// TwinCAT 3 PLC project Untitled1
// ProgramVersion: 3.1.4026.17
// libraries:
//   Tc2_Standard, * (Beckhoff Automation GmbH)
//   Tc2_System, * (Beckhoff Automation GmbH)
//   Tc2_Utilities, * (Beckhoff Automation GmbH)
//   Tc3_EventLogger, * (Beckhoff Automation GmbH)
// project tree:
//   / PlcTask.TcTTO
//   POUs/ Batch.TcPOU, MAIN.TcPOU
// real-time tasks:
//   TASK PlcTask: cycle T#10ms, priority 20, ADS port 350
// I/O:
//   DEVICE Device 2 (EtherCAT) (disabled), AmsNetId 10.12.64.53.3.1
//     Term 1 (EK1100) [EK1100 EtherCAT Coupler (2A E-Bus)]
//       Term 2 (EL1018) [EL1018 8Ch. Dig. Input 24V, 10µs]
//       Term 3 (EL1382) [EL1382 2Ch. Dig. Input thermistor]
//       Term 4 (EL6070-0033) [EL6070-0033 1Ch. Licence key terminal, individual licences]
//       Term 5 (EL6900) [EL6900, TwinSAFE PLC]
//       Term 6 (EL1918) [EL1918, 8Ch. Safety Input 24V, TwinSAFE]
//         modules: Module 1 (FSOE), Module 2 (FSLOGIC)
//       Term 7 (EL9011) [EL9011 End Terminal]

CONFIGURATION Untitled1
    RESOURCE PLC ON TwinCAT3
        TASK PlcTask(INTERVAL := T#10ms, PRIORITY := 20);
        PROGRAM MAIN WITH PlcTask : MAIN;
    END_RESOURCE
END_CONFIGURATION

// ---- POUs/MAIN.TcPOU
PROGRAM MAIN
VAR
	
bInit : BOOL := TRUE; 
    bSend : BOOL := TRUE; 

    fbMsg : FB_TcMessage; 
	{attribute 'TcRpcEnable'} 
	MOVE1 : BOOL;
	
	test : BOOL;
	{ attribute 'TcHmiSymbol.AddSymbol' }
_i       : INT;
	
	{ attribute 'TcHmiSymbol.AddSymbol' }
	numericInputValue : INT;
	
	floattest : REAL;
	dintTest : DINT;

	realValue : REAL;
	
	a : INT;
	
	b : INT;
	
	BSOD : BOOL;
	
END_VAR

IF bInit THEN
    bInit := FALSE; 
    fbMsg.CreateEx(TC_EVENTS.EventTest.Help, 0); 
	fbMsg.CreateEx(TC_EVENTS.EventTest.Help2, 0);
	//fbMsg.CreateEx(TC_EVENTS.EventTest.Help3, 0);
END_IF

IF bSend THEN 
    bSend := FALSE; 
    fbMsg.Send(0); 
END_IF


numericInputValue := 50;

Batch();


IF BSOD THEN 
	numericInputValue := a/b;
END_IF

END_PROGRAM

// ---- POUs/Batch.TcPOU
PROGRAM Batch
VAR
	fbRunBat						: NT_StartProcess;
	NT_StartProcess_Busy			: BOOL;
	NT_StartProcess_Err				: BOOL;
	NT_StartProcess_ErrId			: UDINT;
	Tmout							: TIME;
	bSuccess						: BOOL;
	bBatFilePath					: T_MaxString;
	sBatDirPath						: T_MaxString;
	sBatCmdLine						: T_MaxString;
	NT_Busy							: BOOL;
	NT_Err							: BOOL;
	NT_ErrID						: UDINT;
	fbLocalAMSNetID					: FB_Getlocalamsnetid;
	
	


	bCopyToUSB: BOOL;
END_VAR

IF 	fbRunBat.START AND NOT NT_Busy THEN 
	bCopyToUSB := FALSE;
	
END_IF


IF bCopyToUSB THEN 
	fbLocalAmsnetID.bExecute := TRUE;
	fbRunBat.NETID := '10.12.64.53.1.1';
	fbRunBat.PATHSTR := 'C:\Users\Administrator\Desktop\test.bat';
	fbRunBat.DIRNAME :='C:\Users\Administrator\Desktop';
	fbRunBat.COMNDLINE := '';
	fbRunBat.TMOUT := T#5S;
	fbRunBat.START := TRUE;
	NT_Busy := fbRunBat.BUSY;
	NT_Err := fbRunBat.ERR;
	NT_ErrID := fbRunBat.ERRID;
	
	
END_IF

END_PROGRAM
